FUNCTION_BLOCK FB_Remote
VAR_INPUT
	feedback			: RemoteFeedback;
END_VAR
VAR_OUTPUT
	control				: RemoteControl;
END_VAR
VAR
	txData				: RemoteFeedback;	
	rxData				: RemoteControl;
	
	ipAddr 				: UDINT;
	remotePort 			: UINT;
	localPort 			: UINT;
	
	udpClient 			: FB_UdpClient(ipAddr, remotePort, localPort, SIZEOF(txData), ADR(txData), SIZEOF(rxData), ADR(rxData));
	
END_VAR



udpClient();

METHOD FB_init : BOOL
VAR_INPUT
	bInitRetains : BOOL; // if TRUE, the retain variables are initialized (warm start / cold start)
	bInCopyCode : BOOL;  // if TRUE, the instance afterwards gets moved into the copy code (online change)
	
	// Contructor arguments
	_ipAddr 			: UDINT;
	_remotePort 		: UINT;
	_localPort 		: UINT;
END_VAR
// Initilize parameters
ipAddr := _ipAddr;
remotePort := _remotePort;
localPort := _localPort;

// Construct FB_UdpClient
udpClient.FB_init(bInitRetains, bInCopyCode, ipAddr, remotePort, localPort, SIZEOF(txData), ADR(txData), SIZEOF(rxData), ADR(rxData));
END_METHOD

END_FUNCTION_BLOCK

(* stored: Version 1.1.0.1, ProductVersion 3.1.4020.12
   POU FB_Remote: Id {26b9ef8a-bd47-4ae3-bad5-31fb25883213}, SpecialFunc None
   Method FB_init: Id {1759a608-ff26-4666-ba56-016a8cefa645} *)
